FUNCTION_BLOCK FB_INICIALIZACIJA
VAR_INPUT
	b_SignalToTrig : BOOL;	
	i_nKorak : INT;
END_VAR
VAR_OUTPUT
	b_GibVIzhodisce : BOOL;
	b_GibVPozicijoCakanjaKosa : BOOL;
END_VAR
VAR
	initEdge: INT;
	CLK: INT;
	korak: INT;
	Q: INT;
	R_initEdge : R_TRIG;
	
END_VAR

//ob pritisku na Init tipko gre v izhodisce
R_initEdge(CLK:=b_SignalToTrig);


CASE korak OF
	0:
		IF R_initEdge.Q AND (i_nKorak <> 50) THEN
		main.iKorak := -1;
		END_IF;
		korak := 10;
	10:
		
		IF (main.iKorak = 50) AND R_initEdge.Q THEN	
			main.iKorakRelativnegaPomika := -1;
		END_IF
	
		IF main.iKorak = 100 THEN
			korak := 0;
		END_IF
	
END_CASE

END_FUNCTION_BLOCK

(* stored: Version 1.1.0.1, ProductVersion 3.1.4024.9
   POU FB_INICIALIZACIJA: Id {0abcf521-4fc1-4e1c-9d15-e8080694b344}, SpecialFunc None *)
